SUBAPPLICATION SRT_RPC_FROM_Remote_QXA_OPC_Adapter (* Geraet B (Station 12, 192.168.1.12): wie SRT_RPC_FROM_Remote_QXA_OPC, aber die 3 SERVER_0-Instanzen + AX_CLIENT_1_0 sind hinter EINEM ASRT_AX_SERVER_0_CLIENT_1_0-Baustein hinter einem einzigen bidirektionalen Adapter-Anschluss gebuendelt; ASRT_AX_AX_SPLIT speist sowohl DigitalOutput_Q1 als auch die SR/Toggle-Flipflop-Logik (ASRT_AX_T_FF_SR_2) - 'SUB style': das Protokoll steckt im MyLib::sys-Composite, nicht in der Resource des Geraets *)
  (* Standard: 61499-2; Description: Copyright (c) 2026 Meisterschulen am Ostbahnhof This program and the accompanying materials are made available under the terms of the Eclipse Public License 2.0 which is available at https://www.eclipse.org/legal/epl-2.0/ SPDX-License-Identifier: EPL-2.0 *)
  (* Version 1.0, 2026-09-04, Franz Höpfinger, Meisterschulen am Ostbahnhof, initial API and implementation and/or initial documentation *)
  PACKAGE MyLib::sys;
  IMPORT logiBUS::io::DQ::logiBUS_DO;
  IMPORT logiBUS::io::DQ::logiBUS_DO_S;
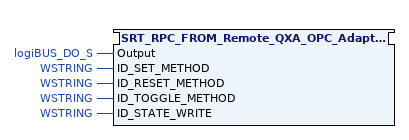
  VAR_INPUT
    Output : logiBUS::io::DQ::logiBUS_DO_S := logiBUS_DO::Invalid; (* Identify the Output Output_Q1..Q8 *)
    ID_SET_METHOD : WSTRING; (* Lokale Methodenadresse (ACTION=CREATE_METHOD) fuer den Set-Methodenaufruf, wird von Geraet A per CALL_METHOD aufgerufen *)
    ID_RESET_METHOD : WSTRING; (* Lokale Methodenadresse (ACTION=CREATE_METHOD) fuer den Reset-Methodenaufruf, wird von Geraet A per CALL_METHOD aufgerufen *)
    ID_TOGGLE_METHOD : WSTRING; (* Lokale Methodenadresse (ACTION=CREATE_METHOD) fuer den Toggle-Methodenaufruf, wird von Geraet A per CALL_METHOD aufgerufen *)
    ID_STATE_WRITE : WSTRING; (* Remote-Ziel-Adresse (BOOL, ACTION=WRITE) fuer den Flipflop-Zustand auf Geraet A *)
  END_VAR
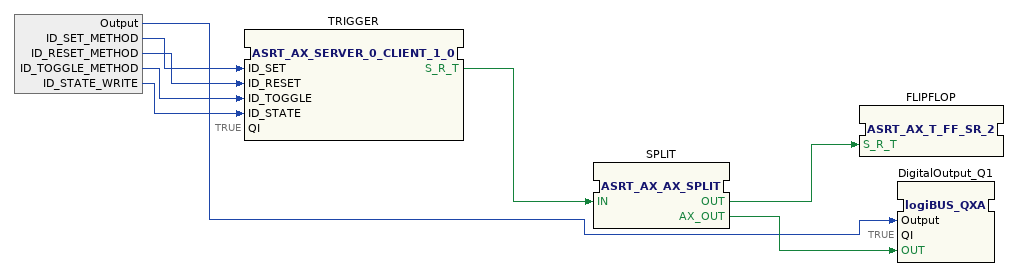
  FBS
    TRIGGER : adapter::net::ASRT_AX_SERVER_0_CLIENT_1_0(QI := TRUE);
    SPLIT : adapter::events::bidirectional::ASRT_AX_AX_SPLIT;
    FLIPFLOP : adapter::events::bidirectional::ASRT_AX_T_FF_SR_2;
    DigitalOutput_Q1 : logiBUS::io::DQ::logiBUS_QXA(QI := TRUE);
  END_FBS
  DATA_CONNECTIONS
    Output TO DigitalOutput_Q1.Output;
    ID_SET_METHOD TO TRIGGER.ID_SET;
    ID_RESET_METHOD TO TRIGGER.ID_RESET;
    ID_TOGGLE_METHOD TO TRIGGER.ID_TOGGLE;
    ID_STATE_WRITE TO TRIGGER.ID_STATE;
  END_CONNECTIONS
  ADAPTER_CONNECTIONS
    TRIGGER.S_R_T TO SPLIT.IN;
    SPLIT.OUT TO FLIPFLOP.S_R_T;
    SPLIT.AX_OUT TO DigitalOutput_Q1.OUT;
  END_CONNECTIONS
END_SUBAPPLICATION
